{attribute 'qualified_only'}
VAR_GLOBAL CONSTANT
	BEEPS_MAX : UINT :=  1971;	
	Beeps : ARRAY[0..BEEPS_MAX] OF REAL := [98, 240, 0, 147, 240, 0, 247, 240, 0, 220, 240, 0, 247, 240, 0, 147, 240, 0, 247, 240, 0, 147, 240, 0, 98, 240, 0, 147, 240, 0, 247, 240, 0, 220, 240, 0, 247, 240, 0, 147, 240, 0, 247, 240, 0, 147, 240, 0, 98, 240, 0, 165, 240, 0, 262, 240, 0, 247, 240, 0, 262, 240, 0, 165, 240, 0, 262, 240, 0, 165, 240, 0, 98, 240, 0, 165, 240, 0, 262, 240, 0, 247, 240, 0, 262, 240, 0, 165, 240, 0, 262, 240, 0, 165, 240, 0, 98, 240, 0, 185, 240, 0, 262, 240, 0, 247, 240, 0, 262, 240, 0, 185, 240, 0, 262, 240, 0, 185, 240, 0, 98, 240, 0, 185, 240, 0, 262, 240, 0, 247, 240, 0, 262, 240, 0, 185, 240, 0, 262, 240, 0, 185, 240, 0, 98, 240, 0, 196, 240, 0, 247, 240, 0, 220, 240, 0, 247, 240, 0, 196, 240, 0, 247, 240, 0, 196, 240, 0, 98, 240, 0, 196, 240, 0, 247, 240, 0, 220, 240, 0, 247, 240, 0, 196, 240, 0, 247, 240, 0, 185, 240, 0, 98, 240, 0, 165, 240, 0, 247, 240, 0, 220, 240, 0, 247, 240, 0, 196, 240, 0, 185, 240, 0, 196, 240, 0, 165, 240, 0, 196, 240, 0, 185, 240, 0, 196, 240, 0, 123, 240, 0, 147, 240, 0, 139, 240, 0, 123, 240, 0, 139, 240, 0, 196, 240, 0, 220, 240, 0, 196, 240, 0, 220, 240, 0, 196, 240, 0, 220, 240, 0, 196, 240, 0, 139, 240, 0, 196, 240, 0, 220, 240, 0, 196, 240, 0, 220, 240, 0, 196, 240, 0, 220, 240, 0, 196, 240, 0, 185, 240, 0, 220, 240, 0, 294, 240, 0, 277, 240, 0, 294, 240, 0, 220, 240, 0, 196, 240, 0, 220, 240, 0, 185, 240, 0, 220, 240, 0, 196, 240, 0, 220, 240, 0, 147, 240, 0, 185, 240, 0, 165, 240, 0, 147, 240, 0, 82, 240, 0, 123, 240, 0, 196, 240, 0, 185, 240, 0, 196, 240, 0, 123, 240, 0, 196, 240, 0, 123, 240, 0, 82, 240, 0, 123, 240, 0, 196, 240, 0, 185, 240, 0, 196, 240, 0, 123, 240, 0, 196, 240, 0, 123, 240, 0, 82, 240, 0, 139, 240, 0, 147, 240, 0, 165, 240, 0, 147, 240, 0, 139, 240, 0, 123, 240, 0, 110, 240, 0, 196, 240, 0, 185, 240, 0, 165, 240, 0, 294, 240, 0, 277, 240, 0, 247, 240, 0, 220, 240, 0, 196, 240, 0, 185, 240, 0, 165, 240, 0, 147, 240, 0, 294, 240, 0, 220, 240, 0, 294, 240, 0, 185, 240, 0, 220, 240, 0, 147, 240, 0, 165, 240, 0, 185, 240, 0, 220, 240, 0, 196, 240, 0, 185, 240, 0, 165, 240, 0, 147, 240, 0, 208, 240, 0, 147, 240, 0, 175, 240, 0, 165, 240, 0, 175, 240, 0, 147, 240, 0, 208, 240, 0, 147, 240, 0, 247, 240, 0, 147, 240, 0, 175, 240, 0, 165, 240, 0, 175, 240, 0, 147, 240, 0, 208, 240, 0, 147, 240, 0, 131, 240, 0, 165, 240, 0, 220, 240, 0, 247, 240, 0, 262, 240, 0, 220, 240, 0, 165, 240, 0, 147, 240, 0, 131, 240, 0, 165, 240, 0, 220, 240, 0, 247, 240, 0, 262, 240, 0, 220, 240, 0, 185, 240, 0, 165, 240, 0, 156, 240, 0, 185, 240, 0, 156, 240, 0, 185, 240, 0, 220, 240, 0, 185, 240, 0, 220, 240, 0, 185, 240, 0, 156, 240, 0, 185, 240, 0, 156, 240, 0, 185, 240, 0, 220, 240, 0, 185, 240, 0, 220, 240, 0, 185, 240, 0, 196, 240, 0, 185, 240, 0, 165, 240, 0, 196, 240, 0, 185, 240, 0, 196, 240, 0, 220, 240, 0, 185, 240, 0, 196, 240, 0, 185, 240, 0, 165, 240, 0, 147, 240, 0, 131, 240, 0, 123, 240, 0, 110, 240, 0, 98, 240, 0, 92, 240, 0, 131, 240, 0, 147, 240, 0, 131, 240, 0, 147, 240, 0, 131, 240, 0, 147, 240, 0, 131, 240, 0, 92, 240, 0, 131, 240, 0, 147, 240, 0, 131, 240, 0, 147, 240, 0, 131, 240, 0, 147, 240, 0, 131, 240, 0, 98, 240, 0, 123, 240, 0, 175, 240, 0, 165, 240, 0, 175, 240, 0, 123, 240, 0, 175, 240, 0, 123, 240, 0, 98, 240, 0, 123, 240, 0, 175, 240, 0, 165, 240, 0, 175, 240, 0, 123, 240, 0, 175, 240, 0, 123, 240, 0, 98, 240, 0, 131, 240, 0, 165, 240, 0, 147, 240, 0, 165, 240, 0, 131, 240, 0, 165, 240, 0, 131, 240, 0, 98, 240, 0, 131, 240, 0, 165, 240, 0, 147, 240, 0, 165, 240, 0, 131, 240, 0, 165, 240, 0, 131, 240, 0, 98, 240, 0, 185, 240, 0, 262, 240, 0, 247, 240, 0, 262, 240, 0, 185, 240, 0, 262, 240, 0, 185, 240, 0, 98, 240, 0, 185, 240, 0, 262, 240, 0, 247, 240, 0, 262, 240, 0, 185, 240, 0, 262, 240, 0, 185, 240, 0, 98, 240, 0, 147, 240, 0, 247, 240, 0, 220, 240, 0, 247, 240, 0, 196, 240, 0, 185, 240, 0, 165, 240, 0, 147, 240, 0, 131, 240, 0, 123, 240, 0, 110, 240, 0, 98, 240, 0, 92, 240, 0, 82, 240, 0, 73, 240, 0, 69, 240, 0, 110, 240, 0, 165, 240, 0, 185, 240, 0, 196, 240, 0, 165, 240, 0, 185, 240, 0, 196, 240, 0, 69, 240, 0, 110, 240, 0, 165, 240, 0, 185, 240, 0, 196, 240, 0, 165, 240, 0, 185, 240, 0, 196, 240, 0, 65, 240, 0, 110, 240, 0, 147, 240, 0, 165, 240, 0, 185, 240, 0, 147, 240, 0, 165, 240, 0, 185, 240, 0, 65, 240, 0, 110, 240, 0, 147, 240, 0, 165, 240, 0, 185, 240, 0, 147, 240, 0, 165, 240, 0, 185, 240, 0, 65, 240, 0, 110, 240, 0, 147, 240, 0, 185, 240, 0, 220, 240, 0, 277, 240, 0, 294, 720, 0, 110, 240, 0, 123, 240, 0, 131, 240, 0, 147, 240, 0, 165, 240, 0, 185, 240, 0, 196, 240, 0, 220, 240, 0, 185, 240, 0, 147, 240, 0, 165, 240, 0, 185, 240, 0, 196, 240, 0, 220, 240, 0, 247, 240, 0, 262, 240, 0, 220, 240, 0, 185, 240, 0, 196, 240, 0, 220, 240, 0, 247, 240, 0, 262, 240, 0, 294, 240, 0, 311, 240, 0, 294, 240, 0, 277, 240, 0, 294, 240, 0, 294, 240, 0, 262, 240, 0, 247, 240, 0, 262, 240, 0, 262, 240, 0, 220, 240, 0, 185, 240, 0, 165, 240, 0, 147, 240, 0, 110, 240, 0, 123, 240, 0, 131, 240, 0, 73, 240, 0, 110, 240, 0, 147, 240, 0, 185, 240, 0, 220, 240, 0, 247, 240, 0, 262, 240, 0, 220, 240, 0, 247, 240, 0, 196, 240, 0, 147, 240, 0, 131, 240, 0, 123, 240, 0, 98, 240, 0, 110, 240, 0, 123, 240, 0, 73, 240, 0, 98, 240, 0, 123, 240, 0, 147, 240, 0, 196, 240, 0, 220, 240, 0, 247, 240, 0, 196, 240, 0, 277, 240, 0, 247, 240, 0, 220, 240, 0, 233, 240, 0, 233, 240, 0, 220, 240, 0, 208, 240, 0, 220, 240, 0, 220, 240, 0, 196, 240, 0, 185, 240, 0, 196, 240, 0, 196, 240, 0, 165, 240, 0, 139, 240, 0, 123, 240, 0, 110, 240, 0, 139, 240, 0, 165, 240, 0, 196, 240, 0, 220, 240, 0, 277, 240, 0, 294, 240, 0, 277, 240, 0, 294, 240, 0, 220, 240, 0, 185, 240, 0, 165, 240, 0, 185, 240, 0, 220, 240, 0, 147, 240, 0, 185, 240, 0, 110, 240, 0, 147, 240, 0, 139, 240, 0, 123, 240, 0, 110, 240, 0, 98, 240, 0, 92, 240, 0, 82, 240, 0, 73, 480, 0, 262, 240, 0, 247, 240, 0, 220, 240, 0, 196, 240, 0, 185, 240, 0, 165, 240, 0, 147, 240, 0, 262, 240, 0, 247, 240, 0, 220, 240, 0, 196, 240, 0, 185, 240, 0, 165, 240, 0, 147, 240, 0, 131, 240, 0, 247, 240, 0, 220, 240, 0, 196, 240, 0, 185, 240, 0, 165, 240, 0, 147, 240, 0, 131, 240, 0, 123, 240, 0, 220, 240, 0, 196, 240, 0, 185, 240, 0, 165, 240, 0, 147, 240, 0, 131, 240, 0, 123, 240, 0, 110, 240, 0, 196, 240, 0, 185, 240, 0, 165, 240, 0, 185, 240, 0, 147, 240, 0, 165, 240, 0, 185, 240, 0, 196, 240, 0, 165, 240, 0, 185, 240, 0, 147, 240, 0, 196, 240, 0, 165, 240, 0, 185, 240, 0, 147, 240, 0, 196, 240, 0, 165, 240, 0, 185, 240, 0, 147, 240, 0, 165, 240, 0, 185, 240, 0, 196, 240, 0, 220, 240, 0, 247, 240, 0, 147, 240, 0, 220, 240, 0, 247, 240, 0, 262, 240, 0, 147, 240, 0, 247, 240, 0, 262, 240, 0, 294, 240, 0, 247, 240, 0, 262, 240, 0, 247, 240, 0, 262, 240, 0, 220, 240, 0, 247, 240, 0, 220, 240, 0, 247, 240, 0, 196, 240, 0, 220, 240, 0, 196, 240, 0, 220, 240, 0, 185, 240, 0, 196, 240, 0, 185, 240, 0, 196, 240, 0, 165, 240, 0, 185, 240, 0, 147, 240, 0, 165, 240, 0, 175, 240, 0, 185, 240, 0, 196, 240, 0, 208, 240, 0, 220, 240, 0, 233, 240, 0, 247, 240, 0, 262, 240, 0, 277, 240, 0, 294, 240, 0, 311, 240, 0, 330, 240, 0, 349, 240, 0, 370, 240, 0, 392, 240, 0, 247, 240, 0, 147, 240, 0, 247, 240, 0, 392, 240, 0, 247, 240, 0, 392, 240, 0, 247, 240, 0, 392, 240, 0, 247, 240, 0, 147, 240, 0, 247, 240, 0, 392, 240, 0, 247, 240, 0, 392, 240, 0, 247, 240, 0, 392, 240, 0, 220, 240, 0, 147, 240, 0, 220, 240, 0, 392, 240, 0, 220, 240, 0, 392, 240, 0, 220, 240, 0, 392, 240, 0, 220, 240, 0, 147, 240, 0, 220, 240, 0, 392, 240, 0, 220, 240, 0, 392, 240, 0, 220, 240, 0, 370, 240, 0, 262, 240, 0, 147, 240, 0, 262, 240, 0, 370, 240, 0, 262, 240, 0, 370, 240, 0, 262, 240, 0, 370, 240, 0, 262, 240, 0, 147, 240, 0, 262, 240, 0, 370, 240, 0, 262, 240, 0, 370, 240, 0, 262, 240, 0, 392, 3840, 0, 220, 240, 0, 220, 240, 0, 220, 240, 0, 220, 240, 0, 220, 240, 0, 220, 240, 0, 220, 240, 0, 220, 240, 0, 220, 240, 0, 220, 240, 0, 220, 240, 0, 220, 240, 0, 220, 240, 0, 220, 240, 0, 220, 240, 0, 220, 240, 0, 220, 240, 0, 220, 240, 0, 220, 240, 0, 220, 240, 0, 220, 240, 0, 220, 240, 0, 220, 240, 0, 220, 240, 0, 220, 240, 0, 220, 240, 0, 220, 240, 0, 220, 240, 0, 220, 240, 0, 220, 240, 0, 220, 240, 0, 220, 240, 0, 220, 240, 0, 220, 240, 0, 220, 240, 0, 220, 240, 0, 220, 240, 0, 220, 240, 0, 220, 240, 0, 220, 240, 0, 220, 240, 0, 220, 240, 0, 220, 240, 0, 220, 240, 0, 220, 240, 0, 220, 240, 0, 220, 240, 0, 147, 240, 0, 147, 240, 0, 147, 240, 0, 147, 240, 0, 147, 240, 0, 147, 240, 0, 147, 240, 0, 147, 240, 0, 147, 240, 0, 147, 240, 0, 147, 240, 0, 147, 240, 0, 147, 240, 0, 147, 240, 0, 247, 3840, 0, 98, 3840, 0, 0, 0, 0];
END_VAR

(* stored: Version 1.1.0.1, ProductVersion 3.1.4019.2
   GVL Bach: Id {0b6d5b88-c0e2-4738-9414-7718c5d4904d} *)
